(* CODESYS project tcl_unittestlibrary.library
   Company: Red Rock Controls Limited
   Description: Lightweight unit test library for TDD
   Version: 1.0.1.0
   Placeholder: tcl_UnitTestLibrary
   Author: Roger Christopher
   Title: tcl_UnitTestLibrary

Project tree, tasks and I/O mapping:
  libraries: Tc2_Standard, * (Beckhoff Automation GmbH); Tc2_System, * (Beckhoff Automation GmbH); Tc2_Utilities, * (Beckhoff Automation GmbH); Tc3_DynamicMemory, * (Beckhoff Automation GmbH); Tc3_Module, * (Beckhoff Automation GmbH)
  Functions/
    function AssertEquals [ST]
    function AssertNearlyEquals [ST]
    function AssertTrue [ST]
  String Utils/
    function FormatString2 [ST]
    function FormatStringEx1 [ST]
    function FormatStringEx2 [ST]
    function block StringSplitter [ST]: GetNext, GetRemainder, HasMore, Init
  Tasks/
    program MAIN [ST]
  Unit Test Framework/
    List Of Tests/
      interface I_ListOfTests: AddTest, Count, GetTest
      function block T_ListOfTests [ST]: AddTest, Clear, FB_exit, FB_init, GetTest, Count
      function block T_TestIterator [ST]: GetNext, HasMore, Initialise
    Test Runner/
      interface I_TestRunner: AddTest
      function block T_TestRunner [ST]: AddTest, ClearTests, Start
    Unit Test/
      function F_LogResult [ST]
      interface I_UnitTest: Init, RunTest, Name
      function block T_UnitTestBase [ST]: FB_init, Init, RunTest, Name
  Unit Tests/
    Unit Tests/
      Assertion Tests/
        function block Test_F_AssertAny_INTS_Differ [ST]: Init, RunTest
        function block TestSuite_AssertTests [ST]
      Example Test/
        function block Test_ExampleTest [ST]: Init, RunTest
      List Of Tests/
        function block Test_GetTestHandlesEmptyList [ST]: Init, Name, RunTest
        function block Test_GetTestHandlesInvalidIndex [ST]: Init, Name, RunTest
        function block Test_GetTestReturnsCorrectTest [ST]: Init, Name, RunTest
        function block Test_IteratorReturnsTests [ST]: Init, Name, RunTest
        function block Test_ListClear [ST]: Init, Name, RunTest
        function block Test_ListCountIncrements [ST]: Init, Name, RunTest
        function block TestSuite_ListOfTests [ST]: AddTest, FB_exit
  Version/
    global variables Global_Version
  global variables Globals
*)

// Version/Global_Version
{attribute 'TcGenerated'}
{attribute 'no-analysis'}
{attribute 'linkalways'}
// This function has been automatically generated from the project information.
VAR_GLOBAL CONSTANT
	{attribute 'const_non_replaced'}
	stLibVersion_tcl_UnitTestLibrary : ST_LibVersion := (iMajor := 1, iMinor := 0, iBuild := 1, iRevision := 0, nFlags := 1, sVersion := '1.0.1.0');
END_VAR

// Globals
{attribute 'qualified_only'}
VAR_GLOBAL

END_VAR

// Functions/AssertEquals
FUNCTION AssertEquals : BOOL
VAR_INPUT
    Source   : T_MaxString;
    Expected : ANY;
    Actual   : ANY;
    Message  : T_MaxString;
END_VAR
VAR_OUTPUT
    Failed : BOOL;
END_VAR
VAR
    ComparisonResult : DINT;
END_VAR

ComparisonResult := MEMCMP(pBuf1 := Expected.pValue,
                           pBuf2 := Actual.pValue,
                           n     := DINT_TO_UDINT(Actual.diSize));

IF Expected.TypeClass <> Actual.TypeClass THEN
    F_LogResult(Source, FormatStringEx1('Assertion Failed - %s', Message));
    Failed := TRUE;
    RETURN;

ELSIF Expected.diSize <> Actual.diSize THEN
    F_LogResult(Source, FormatStringEx1('Assertion Failed - %s', Message));
    Failed := TRUE;
    RETURN;

ELSIF ComparisonResult <> 0 THEN
    F_LogResult(Source, FormatStringEx1('Assertion Failed - %s', Message));
    Failed := TRUE;
    RETURN;
END_IF

AssertEquals := TRUE;

END_FUNCTION

// Unit Test Framework/Unit Test/F_LogResult
FUNCTION F_LogResult : BOOL
VAR_INPUT
    Source  : T_MaxString;
    Message : T_MaxString;
END_VAR
VAR
END_VAR

ADSLOGSTR(msgCtrlMask := ADSLOG_MSGTYPE_STRING OR ADSLOG_MSGTYPE_ERROR OR ADSLOG_MSGTYPE_LOG,
          msgFmtStr   := FormatStringEx2('%s : %s', Source, Message),
          strArg      := '');

END_FUNCTION

// String Utils/FormatStringEx2
{attribute 'hide'}
FUNCTION INTERNAL FormatStringEx2 : T_MaxString
VAR_INPUT
	Format	: T_MaxString;
	arg1	: T_MaxString;
	arg2	: T_MaxString;
END_VAR
VAR
    FB_FormatString1 : FB_FormatString;
END_VAR

FB_FormatString1(
	sFormat:= Format, 
	arg1:= F_STRING(arg1), 
	arg2:= F_STRING(arg2),
	arg3:= , 
	arg4:= , 
	arg5:= , 
	arg6:= , 
	arg7:= , 
	arg8:= , 
	arg9:= , 
	arg10:= , 
	bError=> , 
	nErrId=> , 
	sOut=> FormatStringEx2);

END_FUNCTION

// String Utils/FormatStringEx1
{attribute 'hide'}
FUNCTION INTERNAL FormatStringEx1 : T_MaxString
VAR_INPUT
	Format	: T_MaxString;
	arg1	: T_MaxString;
END_VAR
VAR
    FB_FormatString1 : FB_FormatString;
END_VAR



FB_FormatString1(
	sFormat:= Format, 
	arg1:= F_STRING(arg1), 
	arg2:= , 
	arg3:= , 
	arg4:= , 
	arg5:= , 
	arg6:= , 
	arg7:= , 
	arg8:= , 
	arg9:= , 
	arg10:= , 
	bError=> , 
	nErrId=> , 
	sOut=> FormatStringEx1);

END_FUNCTION

// Functions/AssertNearlyEquals
FUNCTION AssertNearlyEquals : BOOL
VAR_INPUT
    Source   : T_MaxString;
    Expected : LREAL;
    Actual   : LREAL;
	Delta : LREAL;
    Message  : T_MaxString;
END_VAR
VAR_OUTPUT
    Failed : BOOL;
END_VAR

IF ABS(Expected - Actual) > Delta THEN
    F_LogResult(Source, FormatStringEx1('Assertion Failed - %s', Message));
    Failed := TRUE;
    RETURN;
END_IF

AssertNearlyEquals := TRUE;

END_FUNCTION

// Functions/AssertTrue
FUNCTION AssertTrue : BOOL
VAR_INPUT
    Source    : T_MaxString;
    Condition : BOOL;
    Message   : T_MaxString;
END_VAR
VAR_OUTPUT
    Failed : BOOL;
END_VAR

IF NOT Condition THEN
    F_LogResult(Source, FormatStringEx1('Assertion Failed - %s', Message));
    Failed := TRUE;
    RETURN;
END_IF

AssertTrue := TRUE;

END_FUNCTION

// String Utils/FormatString2
{attribute 'hide'}
FUNCTION INTERNAL FormatString2 : T_MaxString
VAR_INPUT
	Format	: T_MaxString;
	arg1	: T_Arg;
	arg2	: T_Arg;
END_VAR
VAR
    FB_FormatString1 : FB_FormatString;
END_VAR

FB_FormatString1(
	sFormat:= Format, 
	arg1:= arg1, 
	arg2:= arg2, 
	arg3:= , 
	arg4:= , 
	arg5:= , 
	arg6:= , 
	arg7:= , 
	arg8:= , 
	arg9:= , 
	arg10:= , 
	bError=> , 
	nErrId=> , 
	sOut=> FormatString2);

END_FUNCTION

// String Utils/StringSplitter
{attribute 'hide'}
FUNCTION_BLOCK INTERNAL StringSplitter
VAR
	SubjectString : TC2_SYSTEM.T_MaxString;
	Delimiter : STRING;
	Delimiter1 : STRING;
	Delimiter2 : STRING;
	NextDelimiterPosition : INT;
	NextDelimiter1Position : INT;
	NextDelimiter2Position : INT;
END_VAR

METHOD GetNext : STRING(255)
VAR_INPUT
END_VAR
VAR
	RemainingLength: INT;
END_VAR
NextDelimiter1Position := FIND(SubjectString , Delimiter1);
NextDelimiter2Position := FIND(SubjectString , Delimiter2);

IF NextDelimiter1Position = 0 THEN
    // use Delimiter 2 position , even if zero...
    NextDelimiterPosition := NextDelimiter2Position;
    Delimiter := Delimiter2;
    
ELSIF NextDelimiter2Position = 0 THEN
    // use Delimiter 1 position , non-zero...
    NextDelimiterPosition := NextDelimiter1Position;
    Delimiter := Delimiter1;

ELSE
    // Both delimters found - use the one nearest the start of the string...
    IF NextDelimiter1Position < NextDelimiter2Position THEN
        NextDelimiterPosition := NextDelimiter1Position;
        Delimiter := Delimiter1;
    ELSE
        NextDelimiterPosition := NextDelimiter2Position;
        Delimiter := Delimiter2;
	END_IF
END_IF

IF NextDelimiterPosition > 0 THEN // delimitter found
    
    // extract next sub-string
	GetNext := LEFT(SubjectString,NextDelimiterPosition - 1);
    
    // remove sub-string from subject string
	RemainingLength := LEN(SubjectString) - NextDelimiterPosition - LEN(Delimiter) + 1;
	SubjectString := RIGHT(SubjectString,RemainingLength);
    
//    // strip any delimitters from front of remaining string
//    WHILE FIND(SubjectString,Delimiter1) = 1 DO
//        SubjectString := RIGHT(SubjectString,LEN(SubjectString) - LEN(Delimiter1));
//	END_WHILE
//    WHILE FIND(SubjectString,Delimiter2) = 1 DO
//        SubjectString := RIGHT(SubjectString,LEN(SubjectString) - LEN(Delimiter2));
//	END_WHILE
ELSE
	GetNext := SubjectString; // return what is left
	SubjectString := '';
END_IF
END_METHOD

METHOD GetRemainder : STRING(255)
GetRemainder := SubjectString; // return what is left
SubjectString := '';
END_METHOD

METHOD HasMore : BOOL
VAR_INPUT
END_VAR
HasMore := SubjectString <> '';
END_METHOD

METHOD Init
VAR_INPUT
		Str : TC2_SYSTEM.T_MaxString;
		Delim1 : STRING;
		Delim2 : STRING;
END_VAR
SubjectString := Str;
NextDelimiterPosition := 0;
Delimiter1 := Delim1;
Delimiter2 := Delim2;
END_METHOD

END_FUNCTION_BLOCK

// Tasks/MAIN
PROGRAM MAIN
VAR
    TestSuite_AssertTests : TestSuite_AssertTests;
    TestSuite_ListOfTests : TestSuite_ListOfTests;
END_VAR

TestSuite_AssertTests();
TestSuite_ListOfTests();

END_PROGRAM

// Unit Tests/Unit Tests/Assertion Tests/TestSuite_AssertTests
{attribute 'analysis' := '-33'} // inhibit unused variable warning
FUNCTION_BLOCK TestSuite_AssertTests
VAR
    TestRunner                : T_TestRunner;
    Test_F_Assert_INTS_Differ : Test_F_AssertAny_INTS_Differ(TestRunner);
END_VAR

TestRunner(TestSuiteName := 'TestSuite_AssertTests');

END_FUNCTION_BLOCK

// Unit Test Framework/Test Runner/T_TestRunner
FUNCTION_BLOCK T_TestRunner IMPLEMENTS I_TestRunner
VAR_INPUT
	TestSuiteName : T_MaxString := 'TestSuite';
    Verbose : BOOL;
END_VAR
VAR
    State : (
        sInit,
        sGetTest,
        sRunTest,
        sCheckResults
    );
    ResultsSummary   : T_MaxString;
    PassedTestsCount : DINT;
    FailedTestsCount : DINT;
    TestList         : T_ListOfTests(Capacity := 50);
    TestIterator     : T_TestIterator;
    CurrentTest      : I_UnitTest;

    RunTests      : BOOL := TRUE;
    TestFailed    : BOOL;
    TestCompleted : BOOL;
END_VAR

CASE State OF
    sInit:
        IF RunTests THEN
            RunTests := FALSE;
            TestIterator.Initialise(TestList);
            ResultsSummary   := '';
            FailedTestsCount := 0;
            PassedTestsCount := 0;
            F_LogResult(Source := TestSuiteName, Message := 'Starting Tests');
            State            := sGetTest;
        END_IF

    sGetTest:
        IF TestIterator.HasMore() THEN
            CurrentTest := TestIterator.GetNext();
            CurrentTest.Init();
            State := sRunTest;
        ELSE
            CurrentTest := 0;
            State       := sCheckResults;
        END_IF

    sRunTest:
        CurrentTest.RunTest(TestCompleted => TestCompleted,
                            TestFailed    => TestFailed);

        IF TestCompleted THEN
            IF TestFailed THEN
                FailedTestsCount := FailedTestsCount + 1;
                F_LogResult(Source := TestSuiteName, Message := FormatStringEx1('Test failed <%s>', CurrentTest.Name));
            ELSE
                PassedTestsCount := PassedTestsCount + 1;
                IF Verbose THEN
                    F_LogResult(Source := TestSuiteName, Message := FormatStringEx1('Test passed <%s>', CurrentTest.Name));
                END_IF
            END_IF
            State := sGetTest;
        END_IF

    sCheckResults:
        ResultsSummary := FormatString2('Tests completed. %d Tests Passed, %d Tests Failed',
                                          F_DINT(PassedTestsCount),
                                          F_DINT(FailedTestsCount));

        F_LogResult(Source  := TestSuiteName,
                    Message := FormatString2('Tests completed. %d Tests Passed, %d Tests Failed',
                                               F_DINT(PassedTestsCount),
                                               F_DINT(FailedTestsCount)));
        State := sInit;

END_CASE

METHOD AddTest
VAR_INPUT
    UnitTest : I_UnitTest;
END_VAR
TestList.AddTest(UnitTest);
END_METHOD

METHOD ClearTests
VAR_INPUT
END_VAR
TestList.Clear();
END_METHOD

{attribute 'call_after_online_change_slot' := '200'}
METHOD Start
VAR_INPUT
END_VAR
RunTests := TRUE;
END_METHOD

END_FUNCTION_BLOCK

// Unit Test Framework/Test Runner/I_TestRunner
INTERFACE I_TestRunner

METHOD AddTest
VAR_INPUT
    UnitTest : I_UnitTest;
END_VAR
END_METHOD

END_INTERFACE

// Unit Test Framework/Unit Test/I_UnitTest
INTERFACE I_UnitTest EXTENDS __SYSTEM.IQueryInterface

METHOD Init
VAR_INPUT
END_VAR
END_METHOD

METHOD FINAL RunTest
VAR_OUTPUT
    TestCompleted : BOOL;
    TestFailed    : BOOL;
END_VAR
END_METHOD

PROPERTY Name : T_MaxString
GET
END_GET
END_PROPERTY

END_INTERFACE

// Unit Test Framework/List Of Tests/T_ListOfTests
FUNCTION_BLOCK T_ListOfTests IMPLEMENTS I_ListOfTests
VAR
    {attribute 'analysis' := '-33'} // inhibit unused variable warning
    DynamicMemoryManager : FB_DynMem_Manager;
    Buffer               : FB_DynMem_Buffer(ipMemMan := DynamicMemoryManager);
    pTest                : POINTER TO I_UnitTest;
    _Count               : DINT;
    Capacity             : DINT;
END_VAR

METHOD AddTest
VAR_INPUT
    Test : I_UnitTest;
END_VAR
IF _Count = Capacity THEN
    Capacity := Capacity * 2;
    Buffer.Resize(nSize     := DINT_TO_UDINT(Capacity) * SIZEOF(PVOID),
                  bPreserve := TRUE,
                  bReset    := FALSE);

    pTest := Buffer.pBuffer;
END_IF

AssertTrue(Source    := 'T_ListOfTests.AddTest()',
             Condition := pTest > 0,
             Message   := 'Buffer not initialised');

IF pTest <> 0 THEN			 
	pTest[_Count] := Test;
	_Count        := _Count + 1;
END_IF
END_METHOD

METHOD Clear
VAR_INPUT
END_VAR
IF pTest = 0 THEN
    // Buffer was not allocated during Fb_init. Try again...
    Buffer.CreateBuffer(nSize  := DINT_TO_UDINT(Capacity) * SIZEOF(PVOID),
                        bReset := TRUE);
END_IF

Buffer.Clear();
_Count := 0;
END_METHOD

METHOD FB_exit : BOOL
VAR_INPUT
    bInCopyCode : BOOL; // if TRUE, the exit method is called for exiting an instance that is copied afterwards (online change).
END_VAR
IF NOT bInCopyCode THEN
    Buffer.DeleteBuffer();
    pTest := 0;
END_IF
END_METHOD

METHOD FB_init : BOOL
VAR_INPUT
    bInitRetains : BOOL; // if TRUE, the retain variables are initialized (warm start / cold start)
    bInCopyCode  : BOOL; // if TRUE, the instance afterwards gets moved into the copy code (online change)
    Capacity     : DINT;
END_VAR
Buffer.CreateBuffer(nSize  := DINT_TO_UDINT(Capacity) * SIZEOF(PVOID),
                    bReset := TRUE);

pTest := Buffer.pBuffer;

THIS^.Capacity := Capacity;
END_METHOD

METHOD GetTest : I_UnitTest
VAR_INPUT
    Index : DINT;
END_VAR
IF Index < _Count AND Index >= 0 THEN
    GetTest := pTest[Index];
END_IF
END_METHOD

PROPERTY Count : DINT
GET
Count := _Count;
END_GET
END_PROPERTY

END_FUNCTION_BLOCK

// Unit Test Framework/List Of Tests/I_ListOfTests
INTERFACE I_ListOfTests

METHOD AddTest
VAR_INPUT
    Test : I_UnitTest;
END_VAR
END_METHOD

PROPERTY Count : DINT
GET
END_GET
END_PROPERTY

METHOD GetTest : I_UnitTest
VAR_INPUT
    Index : DINT;
END_VAR
END_METHOD

END_INTERFACE

// Unit Test Framework/List Of Tests/T_TestIterator
FUNCTION_BLOCK T_TestIterator
VAR_INPUT
END_VAR
VAR_OUTPUT
END_VAR
VAR
    List  : I_ListOfTests;
    Index : DINT;
END_VAR

METHOD GetNext : I_UnitTest
VAR_INPUT
END_VAR
IF List <> 0 AND_THEN HasMore() THEN
    GetNext := List.GetTest(Index);
    Index   := Index + 1;
END_IF
END_METHOD

METHOD HasMore : BOOL
VAR_INPUT
END_VAR
HasMore := List <> 0 AND_THEN (Index < List.Count and List.Count > 0);
END_METHOD

METHOD Initialise : BOOL
VAR_INPUT
    List : I_ListOfTests;
END_VAR
THIS^.List := List;
Index      := 0;
END_METHOD

END_FUNCTION_BLOCK

// Unit Tests/Unit Tests/Assertion Tests/Test_F_AssertAny_INTS_Differ
FUNCTION_BLOCK Test_F_AssertAny_INTS_Differ EXTENDS T_UnitTestBase

METHOD Init
END_METHOD

METHOD RunTest
VAR_OUTPUT
    TestCompleted : BOOL;
    TestFailed    : BOOL;
END_VAR
VAR
    TestValue : INT;
    Actual    : INT;
END_VAR
TestValue := 133;
Actual    := 133;

AssertEquals(Source   := THIS^.TestName,
             Expected := TestValue,
             Actual   := Actual,
             Message  := 'Unexpected value of TestValue',
             Failed   => TestFailed);

TestCompleted := TRUE;
END_METHOD

END_FUNCTION_BLOCK

// Unit Test Framework/Unit Test/T_UnitTestBase
{attribute 'reflection'}
FUNCTION_BLOCK T_UnitTestBase IMPLEMENTS I_UnitTest
VAR_INPUT
END_VAR
VAR_OUTPUT
END_VAR
VAR
    {attribute 'instance-path'}
    {attribute 'no_init'}
    InstanceName : T_MaxString; // Automatically initialised with the full name of the instance
    TestName     : T_MaxString;
    TestRunner   : I_TestRunner;
END_VAR

METHOD FB_init : BOOL
VAR_INPUT
    bInitRetains : BOOL; // if TRUE, the retain variables are initialized (warm start / cold start)
    bInCopyCode  : BOOL; // if TRUE, the instance afterwards gets moved into the copy code (online change)
    TestRunner   : I_TestRunner;
END_VAR
VAR
    StringSplitter : StringSplitter;
END_VAR
StringSplitter.Init(Str    := InstanceName,
                    Delim1 := '.',
                    Delim2 := '');

WHILE StringSplitter.HasMore() DO
    TestName := StringSplitter.GetNext(); // to get last sub-section
END_WHILE

IF TestRunner <> 0 THEN
	THIS^.TestRunner := TestRunner;
	TestRunner.AddTest(THIS^);
END_IF
END_METHOD

METHOD Init
END_METHOD

{attribute 'analysis' := '-33'} // inhibit unused variable warning
METHOD RunTest
VAR_OUTPUT
    TestCompleted : BOOL;
    TestFailed    : BOOL;
END_VAR
END_METHOD

PROPERTY Name : T_MaxString
GET
Name := TestName;
END_GET
END_PROPERTY

END_FUNCTION_BLOCK

// Unit Tests/Unit Tests/List Of Tests/TestSuite_ListOfTests
{attribute 'analysis' := '-33'} // inhibit unused variable warning
FUNCTION_BLOCK TestSuite_ListOfTests
VAR
    TestRunner                      : T_TestRunner;
    Test_GetTestHandlesEmptyList    : Test_GetTestHandlesEmptyList(TestRunner);
    Test_GetTestHandlesInvalidIndex : Test_GetTestHandlesInvalidIndex(TestRunner);
    Test_GetTestReturnsCorrectTest  : Test_GetTestReturnsCorrectTest(TestRunner);
    Test_IteratorReturnsTests       : Test_IteratorReturnsTests(TestRunner);
    Test_ListCountIncrements        : Test_ListCountIncrements(TestRunner);
    Test_ListClear                  : Test_ListClear(TestRunner);
END_VAR

TestRunner(TestSuiteName := 'TestSuite_ListOfTests');

METHOD AddTest
VAR_INPUT
	UnitTest	: I_UnitTest;
END_VAR
TestRunner.AddTest(UnitTest);
END_METHOD

METHOD FB_exit : BOOL
VAR_INPUT
	bInCopyCode : BOOL; // if TRUE, the exit method is called for exiting an instance that is copied afterwards (online change).
END_VAR
TestRunner.ClearTests();
END_METHOD

END_FUNCTION_BLOCK

// Unit Tests/Unit Tests/List Of Tests/Test_GetTestHandlesEmptyList
FUNCTION_BLOCK Test_GetTestHandlesEmptyList EXTENDS T_UnitTestBase IMPLEMENTS I_UnitTest
VAR
    List : T_ListOfTests(Capacity := 10);
END_VAR

METHOD Init
List.Clear();
END_METHOD

PROPERTY Name : Tc2_System.T_MaxString
GET
END_GET
END_PROPERTY

METHOD RunTest
VAR_OUTPUT
    TestCompleted : BOOL;
    TestFailed    : BOOL;
END_VAR
VAR_INST
    TestNumber2 : I_UnitTest;
END_VAR
TestNumber2 := List.GetTest(2);

AssertTrue(Source    := TestName,
             Condition := (TestNumber2 = 0),
             Message   := 'Interface pointer TestNumber2 was not zero',
             Failed    => TestFailed);

TestCompleted := TRUE;
END_METHOD

END_FUNCTION_BLOCK

// Unit Tests/Unit Tests/List Of Tests/Test_GetTestHandlesInvalidIndex
FUNCTION_BLOCK Test_GetTestHandlesInvalidIndex EXTENDS T_UnitTestBase
VAR
    List : T_ListOfTests(Capacity := 10);
END_VAR

METHOD Init
List.Clear();
END_METHOD

PROPERTY Name : Tc2_System.T_MaxString
GET
END_GET
END_PROPERTY

METHOD RunTest
VAR_OUTPUT
    TestCompleted : BOOL;
    TestFailed    : BOOL;
END_VAR
VAR_INST
    TestNumber4 : I_UnitTest;
END_VAR
TestNumber4 := List.GetTest(4);

AssertTrue(Source    := TestName,
             Condition := (TestNumber4 = 0),
             Message   := 'GetTest() has unexpected return value',
             Failed    => TestFailed);

TestCompleted := TRUE;
END_METHOD

END_FUNCTION_BLOCK

// Unit Tests/Unit Tests/List Of Tests/Test_GetTestReturnsCorrectTest
FUNCTION_BLOCK Test_GetTestReturnsCorrectTest EXTENDS T_UnitTestBase
VAR
    List  : T_ListOfTests(Capacity := 10);
    Test0 : Test_ExampleTest(0);
    Test1 : Test_ExampleTest(0);
    Test2 : Test_ExampleTest(0);
    Test3 : Test_ExampleTest(0);
END_VAR

METHOD Init
List.Clear();

List.AddTest(Test0);
List.AddTest(Test1);
List.AddTest(Test2);
List.AddTest(Test3);
END_METHOD

PROPERTY Name : Tc2_System.T_MaxString
GET
END_GET
END_PROPERTY

METHOD RunTest
VAR_OUTPUT
    TestCompleted : BOOL;
    TestFailed    : BOOL;
END_VAR
VAR_INST
    Test2_InterfacePointer : I_UnitTest;
    ReturnValue            : I_UnitTest;
END_VAR
Test2_InterfacePointer := Test2;
ReturnValue            := List.GetTest(2);

AssertEquals(Source   := TestName,
               Expected := Test2_InterfacePointer,
               Actual   := ReturnValue,
               Message  := 'Interface pointer TestNumber2 was not correct',
               Failed   => TestFailed);

TestCompleted := TRUE;
END_METHOD

END_FUNCTION_BLOCK

// Unit Tests/Unit Tests/Example Test/Test_ExampleTest
FUNCTION_BLOCK Test_ExampleTest EXTENDS T_UnitTestBase

METHOD Init
END_METHOD

METHOD RunTest
VAR_OUTPUT
    TestCompleted : BOOL;
    TestFailed    : BOOL;
END_VAR
VAR
    TestValue : LREAL := 133.456;
END_VAR
AssertNearlyEquals(Source   := THIS^.TestName,
                   Expected := 133.456,
                   Actual   := TestValue,
                   Delta    := 0.001,
                   Message  := 'TestValue <> 133.456',
                   Failed   => TestFailed);

TestCompleted := TRUE;
END_METHOD

END_FUNCTION_BLOCK

// Unit Tests/Unit Tests/List Of Tests/Test_IteratorReturnsTests
FUNCTION_BLOCK Test_IteratorReturnsTests EXTENDS T_UnitTestBase
VAR
    List     : T_ListOfTests(Capacity := 10);
    Iterator : T_TestIterator;
    Test0 : Test_ExampleTest(0);
    Test1 : Test_ExampleTest(0);
    Test2 : Test_ExampleTest(0);
    Test3 : Test_ExampleTest(0);
END_VAR

METHOD Init
List.Clear();

List.AddTest(Test0);
List.AddTest(Test1);
List.AddTest(Test2);
List.AddTest(Test3);
END_METHOD

PROPERTY Name : Tc2_System.T_MaxString
GET
END_GET
END_PROPERTY

METHOD RunTest
VAR_OUTPUT
    TestCompleted : BOOL;
    TestFailed    : BOOL;
END_VAR
VAR_INST
    Test2_InterfacePointer : I_UnitTest;
    ReturnValue            : I_UnitTest;
END_VAR
Iterator.Initialise(List);
Iterator.GetNext();
Iterator.GetNext();

Test2_InterfacePointer := Test2;
ReturnValue            := Iterator.GetNext();

AssertEquals(Source   := TestName,
               Expected := Test2_InterfacePointer,
               Actual   := ReturnValue,
               Message  := 'Interface pointer TestNumber2 was not correct',
               Failed   => TestFailed);

TestCompleted := TRUE;
END_METHOD

END_FUNCTION_BLOCK

// Unit Tests/Unit Tests/List Of Tests/Test_ListCountIncrements
FUNCTION_BLOCK Test_ListCountIncrements EXTENDS T_UnitTestBase
VAR
    List  : T_ListOfTests(Capacity := 10);
    Test0 : Test_ExampleTest(0);
END_VAR

METHOD Init
List.Clear();
List.AddTest(Test0);
END_METHOD

PROPERTY Name : Tc2_System.T_MaxString
GET
END_GET
END_PROPERTY

METHOD RunTest
VAR_OUTPUT
    TestCompleted : BOOL;
    TestFailed    : BOOL;
END_VAR
AssertTrue(Source    := TestName,
             Condition := List.Count = 1,
             Message   := 'List.Count was not 1',
             Failed    => TestFailed);

TestCompleted := TRUE;
END_METHOD

END_FUNCTION_BLOCK

// Unit Tests/Unit Tests/List Of Tests/Test_ListClear
FUNCTION_BLOCK Test_ListClear EXTENDS T_UnitTestBase
VAR
    List  : T_ListOfTests(Capacity := 10);
    Test0 : Test_ExampleTest(0);
    Test1 : Test_ExampleTest(0);
    Test2 : Test_ExampleTest(0);
    Test3 : Test_ExampleTest(0);
END_VAR

METHOD Init
List.Clear();
List.AddTest(Test0);
List.AddTest(Test1);
List.AddTest(Test2);
List.AddTest(Test3);
END_METHOD

PROPERTY Name : Tc2_System.T_MaxString
GET
END_GET
END_PROPERTY

METHOD RunTest
VAR_OUTPUT
    TestCompleted : BOOL;
    TestFailed    : BOOL;
END_VAR
AssertTrue(Source    := TestName,
             Condition := List.Count = 4,
             Message   := 'List.Count was not 4',
             Failed    => TestFailed);
			 
List.Clear();			 

AssertTrue(Source    := TestName,
             Condition := List.Count = 0,
             Message   := 'List.Count was not 0',
             Failed    => TestFailed);

TestCompleted := TRUE;
END_METHOD

END_FUNCTION_BLOCK
